{attribute 'linkalways'} 
{attribute 'no_explicit_call' := 'This FB is a CLASS and must be accessed using methods or properties'}
{attribute 'enable_dynamic_creation'}
FUNCTION_BLOCK FINAL LE_SINT EXTENDS Node
VAR
	in1 : _SINT(0);
	in2 : _SINT(0);
	out : _BOOL(FALSE);
END_VAR

METHOD PUBLIC Clone : I_Node
VAR
	pNode : POINTER TO LE_SINT;
END_VAR
pNode := __NEW(LE_SINT);
Clone := pNode^;
END_METHOD

METHOD FB_init : BOOL
VAR_INPUT
	bInitRetains : BOOL; // if TRUE, the retain variables are initialized (warm start / cold start)
	bInCopyCode : BOOL;  // if TRUE, the instance afterwards gets moved into the copy code (online change)
END_VAR
AddInput('in1',THIS^.in1);
AddInput('in2',THIS^.in2);
AddOutput('out', THIS^.out);
END_METHOD

METHOD PROTECTED OnExecute
VAR
END_VAR
out.Value := in1.Value <= in2.Value;
END_METHOD

END_FUNCTION_BLOCK

(* stored: Version 1.1.0.1, ProductVersion 3.1.4024.15
   POU LE_SINT: Id {377b0724-ebc0-411b-9e59-ac02701b2467}, SpecialFunc None
   Folder Constructor: Id {a7797c7a-861a-417e-952d-ac7a8fcade15}
   Method Clone: Id {74eb20bf-2661-4341-a59b-4f80559df814}
   Method FB_init: Id {b6a06f79-217d-40a1-9dd2-9568b56c19de}
   Method OnExecute: Id {e993976e-59c3-42a6-85c6-794236ce13a6} *)
